{attribute addProperty BoxType "EK1122-0000-0018"}
{attribute addProperty Id "Beckhoff_AX2xxxsub_EK1100EK1100_179A0949162A_0001_AX2000_B110_0000AX2000_9B833B5A21627"}
{attribute addProperty CRC "4170803191"}
{attribute addProperty SizeInBites "232"}
{attribute addProperty SizeInBytes "29"}
TYPE Beckhoff_AX2xxxEK1122_F89967F7 EXTENDS EK1122_179A0949 :
STRUCT
	{attribute addProperty Name "Beckhoff_AX2xxxsub_EK1100"}
	Beckhoff_AX2xxxsub_EK1100 : EK1100_179A0949;
	{attribute addProperty Name "A_0001_AX2000_B110_0000"}
	A_0001_AX2000_B110_0000 : AX2000_9B833B5A;
END_STRUCT
END_TYPE

(* stored: Version 1.2.0.0, ProductVersion 3.1.4024.9
   DUT Beckhoff_AX2xxxEK1122_F89967F7: Id {8bfc5d51-b4f8-42b0-9f84-8a7f7dd5cfd7} *)
